PROGRAM P_AP1_Check
VAR_INPUT
	//
	// INT 
	n_Step: INT := 0;	
END_VAR
VAR
	//
	// BOOL 
	b_Condition: BOOL;

	//
	// Timer
	t_AP1_Calibration_Time: TON; 
	
END_VAR

//***********************************************************************************
//
// ETH Zürich / Robotic Fabrication Lab
// HIB C 13 / Stefano-Franscini-Platz 1
// CH-8093 Zürich
// 
// ***********************************************************************************
// 
// PROJECT     :  A061 Inline Mixer
// 
// FUNCTION    :  Step chain for accelerator pump calibration
// 
// AUTHOR      :  Seyma Gürel / Philippe Fleischmann / Weiting Chen
// 
// EMAIL       :  sguerel@ethz.ch / fleischmann@arch.ehtz.ch
// 
// Copyright   :  ETH Zürich (CH) 2021
//
// ***********************************************************************************

//
// Initalization
IF n_Step=0 THEN
	//
	// Check condition 
	b_Condition:=TRUE;
	//
	// Do step
	IF b_Condition THEN
		b_Condition:=FALSE;
		n_Step:=10;
	END_IF
END_IF

//
// Wait for activating calibration
IF n_Step=10 THEN
	//
	// Check condition 
	b_Condition:= GVL_ResearchData.b_RED_Acceleration_Pump_Check_On;
	//
	// Do step
	IF b_Condition THEN
		b_Condition:=FALSE;
		n_Step:=20;
	END_IF
END_IF

//
// Wait for start 
IF n_Step=20 THEN
	//
	// Check condition 
	b_Condition:=GVL_IO.ib_AP1_Ready AND (GVL_IO.ib_AP1_Button_On OR GVL_ResearchData.b_RED_Accelerastor_Pump_Power_On_Laptop);
	//
	// Do step
	IF b_Condition THEN
		b_Condition:=FALSE;
		n_Step:=30;
	END_IF
END_IF

//
// Run calibration until time is over 
IF n_Step=30 THEN
	//
	// Check condition 
	b_Condition:=t_AP1_Calibration_Time.Q; 
	//
	// Do step
	IF b_Condition THEN
		b_Condition:=FALSE;
		n_Step:=40;
	END_IF
END_IF

//
// Return to step 10 
IF n_Step=40 THEN
	//
	// Check condition 
	b_Condition:=TRUE;
	//
	// Do step
	IF b_Condition THEN
		b_Condition:=FALSE;
		//
		// Reset Check 
		GVL_ResearchData.b_RED_Acceleration_Pump_Check_On:=FALSE;
		// Turn off the pump
		GVL_ResearchData.b_RED_Accelerastor_Pump_Power_On_Laptop:=FALSE;
		n_Step:=10;
	END_IF
END_IF

// ****************************************
// Timer
// ****************************************
t_AP1_Calibration_Time(
	IN:=n_Step=30,
	PT:=GVL_ResearchData.n_RED_Acceleration_Pump_Check_Duration);

// ****************************************
// Reset
// ****************************************

IF NOT GVL_ResearchData.b_RED_Acceleration_Pump_Check_On THEN
  //
  // Rest step chain
  n_Step:=0;
END_IF

END_PROGRAM

(* stored: Version 1.1.0.1, ProductVersion 3.1.4024.11
   POU P_AP1_Check: Id {d1e3f63a-2203-42a3-a5b1-25305ed70471}, SpecialFunc None *)
